// TIA Portal project "assembly_system" (V16)

(* hardware
DEVICE "ET 200SP station_1"  ET 200SP-Station
   slot 0: "IO device_1"  IM 155-6 PN/2 HF  6ES7 155-6AU01-0CN0  V4.2
   slot 0: "Rack_0"  Rack  6ES5 710-8MAx1
   slot 1: "DI 8x24VDC HF_1"  DI 8x24VDC HF  6ES7 131-6BF00-0CA0  V2.0
      slot 1: "DI 8x24VDC HF_1"  DI 8x24VDC HF
   slot 2: "DI 8x24VDC HF_2"  DI 8x24VDC HF  6ES7 131-6BF00-0CA0  V2.0
      slot 1: "DI 8x24VDC HF_2"  DI 8x24VDC HF
   slot 3: "DI 8x24VDC HF_3"  DI 8x24VDC HF  6ES7 131-6BF00-0CA0  V2.0
      slot 1: "DI 8x24VDC HF_3"  DI 8x24VDC HF
   slot 4: "DQ 8x24VDC/0.5A HF_1"  DQ 8x24VDC/0.5A HF  6ES7 132-6BF00-0CA0  V2.0
      slot 1: "DQ 8x24VDC/0.5A HF_1"  DQ 8x24VDC/0.5A HF
   slot 5: "DQ 8x24VDC/0.5A HF_2"  DQ 8x24VDC/0.5A HF  6ES7 132-6BF00-0CA0  V2.0
      slot 1: "DQ 8x24VDC/0.5A HF_2"  DQ 8x24VDC/0.5A HF
   slot 6: "Server module_1"  Server module  6ES7 193-6PA00-0AA0  V1.1
      slot 1: "Server module_1"  Server module
   slot 127: "BA 2xRJ45"  BA 2xRJ45  6ES7 193-6AR00-0AA0  V0.0
      slot 1: "Port_1"  X1 P1 R  6ES7 193-6AR00-0AA0  V0.0
      slot 2: "Port_2"  X1 P2 R  6ES7 193-6AR00-0AA0  V0.0
DEVICE "S7-1200 station_1"  S7-1200 Station
   slot 0: "Rack_0"  S7-1200 Rack  Rack  V1.0
   slot 1: "PLC_1"  CPU 1214C DC/DC/DC  6ES7 214-1AG40-0XB0  V4.4
DEVICE "SCALANCE X005"  SCALANCE X-Station
   slot 0: "Switch_1"  6GK5 005-0BA00-1AB2  V1.0
   slot 0: "SCALANCE X rack"  Rail
*)

// ===== PLC "PLC_1"  CPU 1214C DC/DC/DC =====

VAR_GLOBAL   // PLC tag table "Default tag table"
   "Tag_1" AT %M98.0 : Bool;
   "Tag_2" AT %M98.1 : Bool;
   "Tag_3" AT %M98.2 : Bool;
   "Clock_Byte" AT %MB200 : Byte;
   "Clock_10Hz" AT %M200.0 : Bool;
   "Clock_5Hz" AT %M200.1 : Bool;
   "Clock_2.5Hz" AT %M200.2 : Bool;
   "Clock_2Hz" AT %M200.3 : Bool;
   "Clock_1.25Hz" AT %M200.4 : Bool;
   "Clock_1Hz" AT %M200.5 : Bool;
   "Clock_0.625Hz" AT %M200.6 : Bool;
   "Clock_0.5Hz" AT %M200.7 : Bool;
   "Tag_4" AT %M10.6 : Bool;
   "System_Byte" AT %MB30 : Byte;
   "FirstScan" AT %M30.0 : Bool;
   "DiagStatusUpdate" AT %M30.1 : Bool;
   "AlwaysTRUE" AT %M30.2 : Bool;
   "AlwaysFALSE" AT %M30.3 : Bool;
END_VAR

VAR_GLOBAL   // PLC tag table "IO_TAGS"
   "START BUTTON  (N.O.) GAUGING" AT %I0.0 : Bool;
   "STOP BUTTON (N.C.) GAUGING" AT %I0.1 : Bool;
   "EMERGENCY STOP BUTTON (N.C.)" AT %I0.2 : Bool;
   "OUTPUT POWER ON (WHITE) GAUGING" AT %I0.3 : Bool;
   "INPUT 1 FROM PREVIOUS STATION GAUGING" AT %I0.4 : Bool;
   "RESET INDEXING STATION" AT %I0.5 : Bool;
   "AUTO INDEXNIG STATION" AT %I0.6 : Bool;
   "INPUT 2 FROM NEXT STATION GAUGING" AT %I0.7 : Bool;
   "RESET/AUTO SWITCH (RESET)" AT %I1.0 : Bool;
   "RESET/AUTO SWITCH (AUTO)" AT %I1.1 : Bool;
   "REJECT CYLINDER 3A RETRACTED GAUGING" AT %I1.2 : Bool;
   "REJECT CYLINDER 3A EXTENDED GAUGING" AT %I1.3 : Bool;
   "TRANSFER CYLINDER 1A RETRACTED GAUGING" AT %I1.4 : Bool;
   "TRANSFER CYLINDER 1A EXTENDED GAUGING" AT %I1.5 : Bool;
   "TRAVERSE IN END OF TRAVEL POSITION" AT %I4.6 : Bool;
   "TRAVERSE IN START OF TRAVEL POSITION" AT %I4.7 : Bool;
   "PART IN HEIGHT MEASURING POSITION" AT %I2.0 : Bool;
   "PART HEIGHT READING" AT %I2.1 : Bool;
   "GAUGING PORT NOT DETECTED (LIGHT SENSOR)" AT %I2.2 : Bool;
   "AUTOMATIC ON  LAMP (GREEN)" AT %Q0.0 : Bool;
   "OUTPUT 1 TO PREVIOUS STATION GAUGING" AT %Q0.1 : Bool;
   "OUTPUT 2 TO PREVIOUS STATION GAUGING" AT %Q0.2 : Bool;
   "OUTPUT 1 TO NEXT STATION GAUGING" AT %Q0.3 : Bool;
   "OUTPUT 2 TO NEXT STATION GAUGING" AT %Q0.4 : Bool;
   "EXTEND REJECT CYLINDER GAUGING" AT %Q0.5 : Bool;
   "EXTEND TRANSFER CYLINDER GAUGING" AT %Q0.6 : Bool;
   "RETRACT TRANSFER CYLINDER GAUGING" AT %Q0.7 : Bool;
   "GAUGING MOTOR STARTER FORWARD" AT %Q1.0 : Bool;
   "GAUGING MOTOR STARTER REVERSE" AT %Q1.1 : Bool;
   "EXTEND LIFT CYLINDER INDEXING" AT %Q3.6 : Bool;
   "AUTOMATIC ON (GREEN)(1)" AT %Q2.0 : Bool;
   "CLOSE GRIPPER 3A(1)" AT %Q3.3 : Bool;
   "EMERGENCY STOP BUTTON (N.C.) INDEXING" AT %I2.5 : Bool;
   "EXTEND LIFT CYLINDER 1A GAUGING" AT %Q2.6 : Bool;
   "EXTEND ROTATION CYLINDER 2A INDEXING" AT %Q3.4 : Bool;
   "EXTEND TRANSFER CYLINDER 3A INDEXING" AT %Q2.5 : Bool;
   "INDEXING TABLE IN HOME POSITION" AT %I4.3 : Bool;
   "INPUT 1 FROM NEXT STATION INDEXING" AT %I3.1 : Bool;
   "INPUT 1 FROM PREVIOUS STATION INDEXING" AT %I2.7 : Bool;
   "INPUT 2 FROM NEXT STATION INDEXING" AT %I3.2 : Bool;
   "INPUT 2 FROM PREVIOUS STATION INDEXING" AT %I3.0 : Bool;
   "LIFT CYLINDER 1A EXTENDED INDEXING" AT %I3.6 : Bool;
   "LIFT CYLINDER 1A RETRACTED INDEXING" AT %I3.5 : Bool;
   "OUTPUT 1 TO NEXT STATION INDEXING" AT %Q2.3 : Bool;
   "OUTPUT 1 TO PREVIOUS STATION INDEXING" AT %Q2.1 : Bool;
   "OUTPUT 2 TO NEXT STATION INDEXING" AT %Q2.4 : Bool;
   "OUTPUT 2 TO PREVIOUS STATION INDEXING" AT %Q2.2 : Bool;
   "OUTPUT POWER ON (WHITE) INDEXING" AT %I2.6 : Bool;
   "PART PRESENT (INITIAL POSITION)" AT %I4.5 : Bool;
   "PART PRESENT (ORIENTATION POSITION)" AT %I3.7 : Bool;
   "RELEASE GRIPPER 3A" AT %Q3.2 : Bool;
   "RETRACT LIFT CYLINDER 1A INDEXING" AT %Q2.7 : Bool;
   "RETRACT ROTATION CYLINDER 2A INDEXING" AT %Q3.5 : Bool;
   "ROTATION CYLINDER 2A EXTENDED INDEXING" AT %I4.1 : Bool;
   "ROTATION CYLINDER 2A RETRACTED INDEXING" AT %I4.0 : Bool;
   "INDEXING SPOOL UPPER PORT DETECTED" AT %I4.2 : Bool;
   "START BUTTON  (N.O.) INDEXING" AT %I2.3 : Bool;
   "STEPPER MOTOR  45°" AT %Q3.0 : Bool;
   "STEPPER MOTOR 90°" AT %Q3.1 : Bool;
   "STEPPER MOTOR READY" AT %I4.4 : Bool;
   "STOP BUTTON (N.C.) INDEXING" AT %I2.4 : Bool;
   "TRANSFER CYLINDER 4A EXTENDED(1)" AT %I3.4 : Bool;
   "TRANSFER CYLINDER 4A RETRACTED(1)" AT %I3.3 : Bool;
END_VAR

DATA_BLOCK "gauging_Modes_data"   // DB1
{ S7_Optimized_Access := 'TRUE' }
VERSION : 0.1
   VAR
      Automatic : Bool;
      Manual : Bool;
      Reset : Bool;
      "Pre-Automatic" : Bool;
   END_VAR
BEGIN
END_DATA_BLOCK

DATA_BLOCK "gauging_outputs_data"   // DB2
{ S7_Optimized_Access := 'TRUE' }
VERSION : 0.1
   VAR
      "Extend reject cylinder" : Bool;
      "Extend transfer cylinder" : Bool;
      "Retract transfer cylinder" : Bool;
      "Motor forward" : Bool;
      "Motor Reverse" : Bool;
      "Extend Lift Cylinder" : Bool;
      Output : Bool;
   END_VAR
BEGIN
END_DATA_BLOCK

DATA_BLOCK "gauging_status_data"   // DB3
{ S7_Optimized_Access := 'TRUE' }
VERSION : 0.1
   VAR
      steps : Int;
      "port not detected" : Bool;
      "height detected" : Bool;
      next_step : Bool;
      input_from_previous_Station : Bool;
   END_VAR
BEGIN
END_DATA_BLOCK

DATA_BLOCK "indexing_Modes_data"   // DB18
{ S7_Optimized_Access := 'TRUE' }
VERSION : 0.1
   VAR
      Automatic : Bool;
      Manual : Bool;
      Reset : Bool;
      "Pre-Automatic" : Bool;
   END_VAR
BEGIN
END_DATA_BLOCK

DATA_BLOCK "indexing_output_data"   // DB19
{ S7_Optimized_Access := 'TRUE' }
VERSION : 0.1
   VAR
      "extend transfer cylinder" : Bool;
      "extend lift cylinder_1" : Bool;
      "extend lift cylinder_2" : Bool;
      "retract lift cylinder_1" : Bool;
      "retract lift cylinder_2" : Bool;
      STEP1_MOTOR_45 : Bool;
      STEP3_MOTOR_45 : Bool;
      STEP4_MOTOR_90 : Bool;
      STEP11_MOTOR_90 : Bool;
      "release gripper" : Bool;
      "close gripper" : Bool;
      "extend rotation" : Bool;
      "retract rotation" : Bool;
      output : Bool;
   END_VAR
BEGIN
END_DATA_BLOCK

DATA_BLOCK "indexing_status_data"   // DB20
{ S7_Optimized_Access := 'TRUE' }
VERSION : 0.1
   VAR
      "CORRECT ORIENTATION" : Bool;
      STEPS : Int;
      next_step : Bool;
      previous_output : Bool;
   END_VAR
BEGIN
END_DATA_BLOCK

// folder: System blocks/Program resources

DATA_BLOCK "port_detection_wait"   // DB4
{ S7_Optimized_Access := 'TRUE' }
AUTHOR : Simatic
FAMILY : IEC
NAME : IEC_TMR
VERSION : 1.0
// stored: InstanceOfName IEC_TIMER
"IEC_TIMER"
BEGIN
END_DATA_BLOCK

DATA_BLOCK "retract_delay"   // DB5
{ S7_Optimized_Access := 'TRUE' }
AUTHOR : Simatic
FAMILY : IEC
NAME : IEC_TMR
VERSION : 1.0
// stored: InstanceOfName IEC_TIMER
"IEC_TIMER"
BEGIN
END_DATA_BLOCK

DATA_BLOCK "next_step_delay"   // DB6
{ S7_Optimized_Access := 'TRUE' }
AUTHOR : Simatic
FAMILY : IEC
NAME : IEC_TMR
VERSION : 1.0
// stored: InstanceOfName IEC_TIMER
"IEC_TIMER"
BEGIN
END_DATA_BLOCK

DATA_BLOCK "height_Timer_0_DB"   // DB7
{ S7_Optimized_Access := 'TRUE' }
AUTHOR : Simatic
FAMILY : IEC
NAME : IEC_TMR
VERSION : 1.0
// stored: InstanceOfName IEC_TIMER
"IEC_TIMER"
BEGIN
END_DATA_BLOCK

DATA_BLOCK "retract_wait"   // DB8
{ S7_Optimized_Access := 'TRUE' }
AUTHOR : Simatic
FAMILY : IEC
NAME : IEC_TMR
VERSION : 1.0
// stored: InstanceOfName IEC_TIMER
"IEC_TIMER"
BEGIN
END_DATA_BLOCK

DATA_BLOCK "next_step_wait_1"   // DB9
{ S7_Optimized_Access := 'TRUE' }
AUTHOR : Simatic
FAMILY : IEC
NAME : IEC_TMR
VERSION : 1.0
// stored: InstanceOfName IEC_TIMER
"IEC_TIMER"
BEGIN
END_DATA_BLOCK

DATA_BLOCK "motor_wait"   // DB10
{ S7_Optimized_Access := 'TRUE' }
AUTHOR : Simatic
FAMILY : IEC
NAME : IEC_TMR
VERSION : 1.0
// stored: InstanceOfName IEC_TIMER
"IEC_TIMER"
BEGIN
END_DATA_BLOCK

DATA_BLOCK "extend_retract_wait"   // DB11
{ S7_Optimized_Access := 'TRUE' }
AUTHOR : Simatic
FAMILY : IEC
NAME : IEC_TMR
VERSION : 1.0
// stored: InstanceOfName IEC_TIMER
"IEC_TIMER"
BEGIN
END_DATA_BLOCK

DATA_BLOCK "wait_Timer"   // DB12
{ S7_Optimized_Access := 'TRUE' }
AUTHOR : Simatic
FAMILY : IEC
NAME : IEC_TMR
VERSION : 1.0
// stored: InstanceOfName IEC_TIMER
"IEC_TIMER"
BEGIN
END_DATA_BLOCK

DATA_BLOCK "motor90_Timer"   // DB13
{ S7_Optimized_Access := 'TRUE' }
AUTHOR : Simatic
FAMILY : IEC
NAME : IEC_TMR
VERSION : 1.0
// stored: InstanceOfName IEC_TIMER
"IEC_TIMER"
BEGIN
END_DATA_BLOCK

DATA_BLOCK "delay_gripper_clamp"   // DB14
{ S7_Optimized_Access := 'TRUE' }
AUTHOR : Simatic
FAMILY : IEC
NAME : IEC_TMR
VERSION : 1.0
// stored: InstanceOfName IEC_TIMER
"IEC_TIMER"
BEGIN
END_DATA_BLOCK

DATA_BLOCK "lift_wait_DB"   // DB15
{ S7_Optimized_Access := 'TRUE' }
AUTHOR : Simatic
FAMILY : IEC
NAME : IEC_TMR
VERSION : 1.0
// stored: InstanceOfName IEC_TIMER
"IEC_TIMER"
BEGIN
END_DATA_BLOCK

DATA_BLOCK "gripper_Timer"   // DB16
{ S7_Optimized_Access := 'TRUE' }
AUTHOR : Simatic
FAMILY : IEC
NAME : IEC_TMR
VERSION : 1.0
// stored: InstanceOfName IEC_TIMER
"IEC_TIMER"
BEGIN
END_DATA_BLOCK

DATA_BLOCK "transfer_delay_DB"   // DB17
{ S7_Optimized_Access := 'TRUE' }
AUTHOR : Simatic
FAMILY : IEC
NAME : IEC_TMR
VERSION : 1.0
// stored: InstanceOfName IEC_TIMER
"IEC_TIMER"
BEGIN
END_DATA_BLOCK

DATA_BLOCK "retract_delay_1"   // DB21
{ S7_Optimized_Access := 'TRUE' }
AUTHOR : Simatic
FAMILY : IEC
NAME : IEC_TMR
VERSION : 1.0
// stored: InstanceOfName IEC_TIMER
"IEC_TIMER"
BEGIN
END_DATA_BLOCK

DATA_BLOCK "retract_DB"   // DB22
{ S7_Optimized_Access := 'TRUE' }
AUTHOR : Simatic
FAMILY : IEC
NAME : IEC_TMR
VERSION : 1.0
// stored: InstanceOfName IEC_TIMER
"IEC_TIMER"
BEGIN
END_DATA_BLOCK

// folder: (top level)

FUNCTION "gauging_modes" : Void   // FC1, LAD
TITLE = Modes Setup
{ S7_Optimized_Access := 'TRUE' }
VERSION : 0.1
BEGIN

REGION Network 1: Automatic Mode
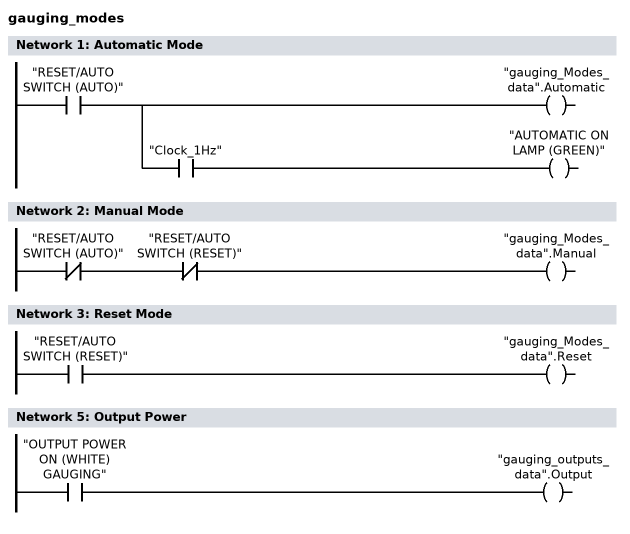
   RUNG wire#powerrail
      Contact( "RESET/AUTO SWITCH (AUTO)" )
      wire#w1
      Coil( "gauging_Modes_data".Automatic )
   END_RUNG
   RUNG wire#w1
      Contact( "Clock_1Hz" )
      Coil( "AUTOMATIC ON  LAMP (GREEN)" )
   END_RUNG
   // the same network as SCL:
   "gauging_Modes_data".Automatic := "RESET/AUTO SWITCH (AUTO)";
   "AUTOMATIC ON  LAMP (GREEN)" := "RESET/AUTO SWITCH (AUTO)" AND "Clock_1Hz";
END_REGION

REGION Network 2: Manual Mode
   RUNG wire#powerrail
      I_Contact( "RESET/AUTO SWITCH (AUTO)" )
      I_Contact( "RESET/AUTO SWITCH (RESET)" )
      Coil( "gauging_Modes_data".Manual )
   END_RUNG
   // the same network as SCL:
   "gauging_Modes_data".Manual := NOT "RESET/AUTO SWITCH (AUTO)" AND NOT "RESET/AUTO SWITCH (RESET)";
END_REGION

REGION Network 3: Reset Mode
   RUNG wire#powerrail
      Contact( "RESET/AUTO SWITCH (RESET)" )
      Coil( "gauging_Modes_data".Reset )
   END_RUNG
   // the same network as SCL:
   "gauging_Modes_data".Reset := "RESET/AUTO SWITCH (RESET)";
END_REGION

REGION Network 4: Pre-Automatic Mode
END_REGION

REGION Network 5: Output Power
   RUNG wire#powerrail
      Contact( "OUTPUT POWER ON (WHITE) GAUGING" )
      Coil( "gauging_outputs_data".Output )
   END_RUNG
   // the same network as SCL:
   "gauging_outputs_data".Output := "OUTPUT POWER ON (WHITE) GAUGING";
END_REGION
END_FUNCTION

FUNCTION "gauging_outputs" : Void   // FC2, LAD
{ S7_Optimized_Access := 'TRUE' }
VERSION : 0.1
BEGIN

REGION Network 1: Gauging Reject Cylinder
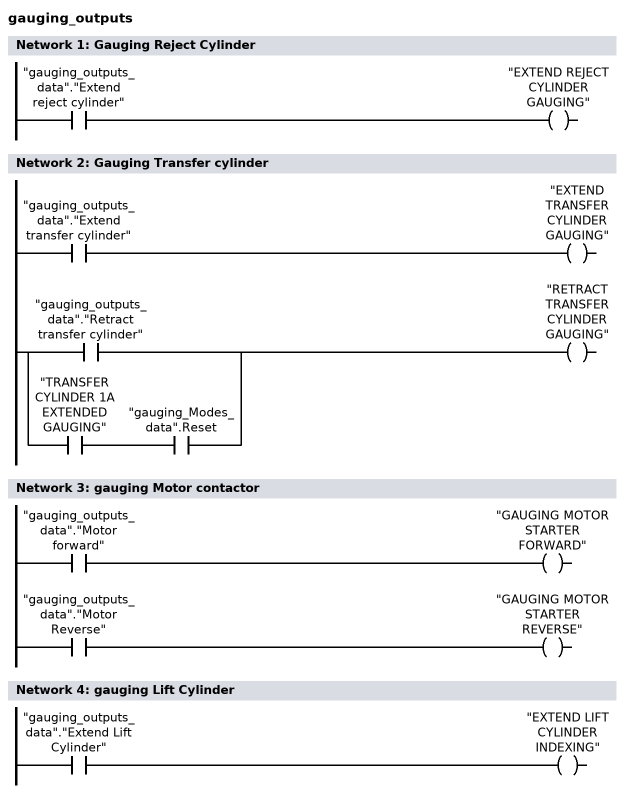
   RUNG wire#powerrail
      Contact( "gauging_outputs_data"."Extend reject cylinder" )
      Coil( "EXTEND REJECT CYLINDER GAUGING" )
   END_RUNG
   // the same network as SCL:
   "EXTEND REJECT CYLINDER GAUGING" := "gauging_outputs_data"."Extend reject cylinder";
END_REGION

REGION Network 2: Gauging Transfer cylinder
   RUNG wire#powerrail
      Contact( "gauging_outputs_data"."Extend transfer cylinder" )
      Coil( "EXTEND TRANSFER CYLINDER GAUGING" )
   END_RUNG
   RUNG wire#powerrail
      Contact( "gauging_outputs_data"."Retract transfer cylinder" )
      wire#w1
      Coil( "RETRACT TRANSFER CYLINDER GAUGING" )
   END_RUNG
   RUNG wire#powerrail
      Contact( "TRANSFER CYLINDER 1A EXTENDED GAUGING" )
      Contact( "gauging_Modes_data".Reset )
   END_RUNG wire#w1
   // the same network as SCL:
   "EXTEND TRANSFER CYLINDER GAUGING" := "gauging_outputs_data"."Extend transfer cylinder";
   "RETRACT TRANSFER CYLINDER GAUGING" := "gauging_outputs_data"."Retract transfer cylinder" OR ("TRANSFER CYLINDER 1A EXTENDED GAUGING" AND "gauging_Modes_data".Reset);
END_REGION

REGION Network 3: gauging Motor contactor
   RUNG wire#powerrail
      Contact( "gauging_outputs_data"."Motor forward" )
      Coil( "GAUGING MOTOR STARTER FORWARD" )
   END_RUNG
   RUNG wire#powerrail
      Contact( "gauging_outputs_data"."Motor Reverse" )
      Coil( "GAUGING MOTOR STARTER REVERSE" )
   END_RUNG
   // the same network as SCL:
   "GAUGING MOTOR STARTER FORWARD" := "gauging_outputs_data"."Motor forward";
   "GAUGING MOTOR STARTER REVERSE" := "gauging_outputs_data"."Motor Reverse";
END_REGION

REGION Network 4: gauging Lift Cylinder
   RUNG wire#powerrail
      Contact( "gauging_outputs_data"."Extend Lift Cylinder" )
      Coil( "EXTEND LIFT CYLINDER INDEXING" )
   END_RUNG
   // the same network as SCL:
   "EXTEND LIFT CYLINDER INDEXING" := "gauging_outputs_data"."Extend Lift Cylinder";
END_REGION
END_FUNCTION

FUNCTION "gauging_utils" : Void   // FC3, LAD
{ S7_Optimized_Access := 'TRUE' }
VERSION : 0.1
   VAR_TEMP   // added for the SCL form of the ladder/FBD networks
      _w1 : Bool;
      _w2 : Bool;
   END_VAR
BEGIN

REGION Network 1: SETUP: output, start, reset
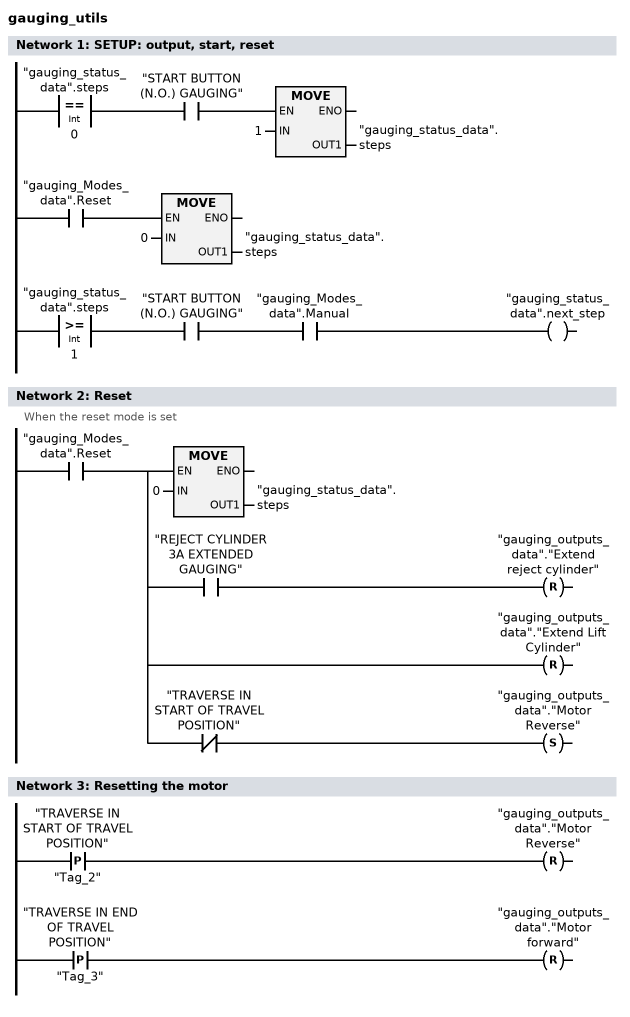
   RUNG wire#powerrail
      { S7_Templates := "SrcType := Int" } EQ_Contact(in1 := "gauging_status_data".steps, in2 := 0)
      Contact( "START BUTTON  (N.O.) GAUGING" )
      Move(in := 1, out1 => "gauging_status_data".steps)
   END_RUNG
   RUNG wire#powerrail
      Contact( "gauging_Modes_data".Reset )
      Move(in := 0, out1 => "gauging_status_data".steps)
   END_RUNG
   RUNG wire#powerrail
      { S7_Templates := "SrcType := Int" } GE_Contact(in1 := "gauging_status_data".steps, in2 := 1)
      Contact( "START BUTTON  (N.O.) GAUGING" )
      Contact( "gauging_Modes_data".Manual )
      Coil( "gauging_status_data".next_step )
   END_RUNG
   // the same network as SCL:
   IF ("gauging_status_data".steps = 0) AND "START BUTTON  (N.O.) GAUGING" THEN
       "gauging_status_data".steps := 1;
   END_IF;
   IF "gauging_Modes_data".Reset THEN "gauging_status_data".steps := 0; END_IF;
   "gauging_status_data".next_step := ("gauging_status_data".steps >= 1) AND "START BUTTON  (N.O.) GAUGING" AND "gauging_Modes_data".Manual;
END_REGION

REGION Network 2: Reset
   // When the reset mode is set
   RUNG wire#powerrail
      Contact( "gauging_Modes_data".Reset )
      wire#w1
      Move(in := 0, out1 => "gauging_status_data".steps)
   END_RUNG
   RUNG wire#w1
      Contact( "REJECT CYLINDER 3A EXTENDED GAUGING" )
      R_Coil( "gauging_outputs_data"."Extend reject cylinder" )
   END_RUNG
   RUNG wire#w1
      R_Coil( "gauging_outputs_data"."Extend Lift Cylinder" )
   END_RUNG
   RUNG wire#w1
      I_Contact( "TRAVERSE IN START OF TRAVEL POSITION" )
      S_Coil( "gauging_outputs_data"."Motor Reverse" )
   END_RUNG
   // the same network as SCL:
   IF "gauging_Modes_data".Reset THEN "gauging_status_data".steps := 0; END_IF;
   IF "gauging_Modes_data".Reset AND "REJECT CYLINDER 3A EXTENDED GAUGING" THEN
       "gauging_outputs_data"."Extend reject cylinder" := FALSE;
   END_IF;
   IF "gauging_Modes_data".Reset THEN "gauging_outputs_data"."Extend Lift Cylinder" := FALSE; END_IF;
   IF "gauging_Modes_data".Reset AND NOT "TRAVERSE IN START OF TRAVEL POSITION" THEN
       "gauging_outputs_data"."Motor Reverse" := TRUE;
   END_IF;
END_REGION

REGION Network 3: Resetting the motor
   RUNG wire#powerrail
      P_Contact(operand := "TRAVERSE IN START OF TRAVEL POSITION", bit := "Tag_2")
      R_Coil( "gauging_outputs_data"."Motor Reverse" )
   END_RUNG
   RUNG wire#powerrail
      P_Contact(operand := "TRAVERSE IN END OF TRAVEL POSITION", bit := "Tag_3")
      R_Coil( "gauging_outputs_data"."Motor forward" )
   END_RUNG
   // the same network as SCL:
   #_w1 := "TRAVERSE IN START OF TRAVEL POSITION" AND NOT "Tag_2";   // rising edge of "TRAVERSE IN START OF TRAVEL POSITION"
   "Tag_2" := "TRAVERSE IN START OF TRAVEL POSITION";
   IF #_w1 THEN "gauging_outputs_data"."Motor Reverse" := FALSE; END_IF;
   #_w2 := "TRAVERSE IN END OF TRAVEL POSITION" AND NOT "Tag_3";   // rising edge of "TRAVERSE IN END OF TRAVEL POSITION"
   "Tag_3" := "TRAVERSE IN END OF TRAVEL POSITION";
   IF #_w2 THEN "gauging_outputs_data"."Motor forward" := FALSE; END_IF;
END_REGION
END_FUNCTION

FUNCTION "gauging_operation" : Void   // FC4, LAD
{ S7_Optimized_Access := 'TRUE' }
VERSION : 0.1
   VAR_TEMP   // added for the SCL form of the ladder/FBD networks
      _w1 : Bool;
   END_VAR
BEGIN

REGION Network 1: Setup
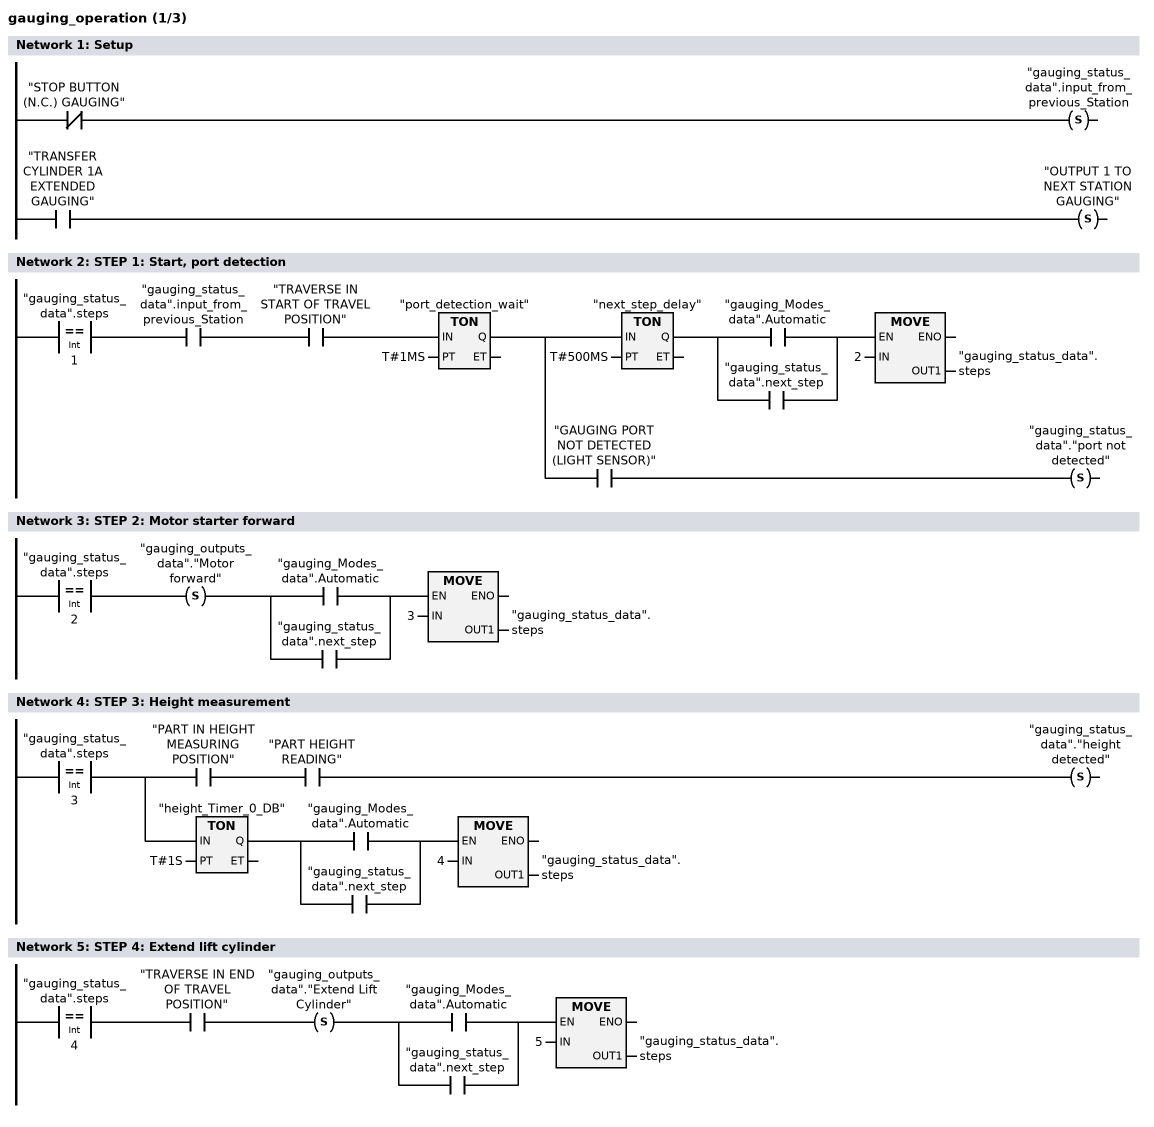
   RUNG wire#powerrail
      I_Contact( "STOP BUTTON (N.C.) GAUGING" )
      S_Coil( "gauging_status_data".input_from_previous_Station )
   END_RUNG
   RUNG wire#powerrail
      Contact( "TRANSFER CYLINDER 1A EXTENDED GAUGING" )
      S_Coil( "OUTPUT 1 TO NEXT STATION GAUGING" )
   END_RUNG
   // the same network as SCL:
   IF NOT "STOP BUTTON (N.C.) GAUGING" THEN
       "gauging_status_data".input_from_previous_Station := TRUE;
   END_IF;
   IF "TRANSFER CYLINDER 1A EXTENDED GAUGING" THEN "OUTPUT 1 TO NEXT STATION GAUGING" := TRUE; END_IF;
END_REGION

REGION Network 2: STEP 1: Start, port detection
   "port_detection_wait".TON(IN := ("gauging_status_data".steps = 1) AND "gauging_status_data".input_from_previous_Station AND "TRAVERSE IN START OF TRAVEL POSITION",
                           PT := T#1MS);
   "next_step_delay".TON(IN := "port_detection_wait".Q, PT := T#500MS);
   IF "next_step_delay".Q AND ("gauging_Modes_data".Automatic OR "gauging_status_data".next_step) THEN
       "gauging_status_data".steps := 2;
   END_IF;
   IF "port_detection_wait".Q AND "GAUGING PORT NOT DETECTED (LIGHT SENSOR)" THEN
       "gauging_status_data"."port not detected" := TRUE;
   END_IF;
END_REGION

REGION Network 3: STEP 2: Motor starter forward
   RUNG wire#powerrail
      { S7_Templates := "SrcType := Int" } EQ_Contact(in1 := "gauging_status_data".steps, in2 := 2)
      S_Coil( "gauging_outputs_data"."Motor forward" )
      wire#w1
      Contact( "gauging_Modes_data".Automatic )
      wire#w2
      Move(in := 3, out1 => "gauging_status_data".steps)
   END_RUNG
   RUNG wire#w1
      Contact( "gauging_status_data".next_step )
   END_RUNG wire#w2
   // the same network as SCL:
   #_w1 := "gauging_status_data".steps = 2;
   IF #_w1 THEN "gauging_outputs_data"."Motor forward" := TRUE; END_IF;
   IF #_w1 AND ("gauging_Modes_data".Automatic OR "gauging_status_data".next_step) THEN
       "gauging_status_data".steps := 3;
   END_IF;
END_REGION

REGION Network 4: STEP 3: Height measurement
   #_w1 := "gauging_status_data".steps = 3;
   IF #_w1 AND "PART IN HEIGHT MEASURING POSITION" AND "PART HEIGHT READING" THEN
       "gauging_status_data"."height detected" := TRUE;
   END_IF;
   "height_Timer_0_DB".TON(IN := #_w1, PT := T#1S);
   IF "height_Timer_0_DB".Q AND ("gauging_Modes_data".Automatic OR "gauging_status_data".next_step) THEN
       "gauging_status_data".steps := 4;
   END_IF;
END_REGION

REGION Network 5: STEP 4: Extend lift cylinder
   RUNG wire#powerrail
      { S7_Templates := "SrcType := Int" } EQ_Contact(in1 := "gauging_status_data".steps, in2 := 4)
      Contact( "TRAVERSE IN END OF TRAVEL POSITION" )
      S_Coil( "gauging_outputs_data"."Extend Lift Cylinder" )
      wire#w1
      Contact( "gauging_Modes_data".Automatic )
      wire#w2
      Move(in := 5, out1 => "gauging_status_data".steps)
   END_RUNG
   RUNG wire#w1
      Contact( "gauging_status_data".next_step )
   END_RUNG wire#w2
   // the same network as SCL:
   #_w1 := ("gauging_status_data".steps = 4) AND "TRAVERSE IN END OF TRAVEL POSITION";
   IF #_w1 THEN "gauging_outputs_data"."Extend Lift Cylinder" := TRUE; END_IF;
   IF #_w1 AND ("gauging_Modes_data".Automatic OR "gauging_status_data".next_step) THEN
       "gauging_status_data".steps := 5;
   END_IF;
END_REGION

REGION Network 6: STEP 5: Check port and height orientation
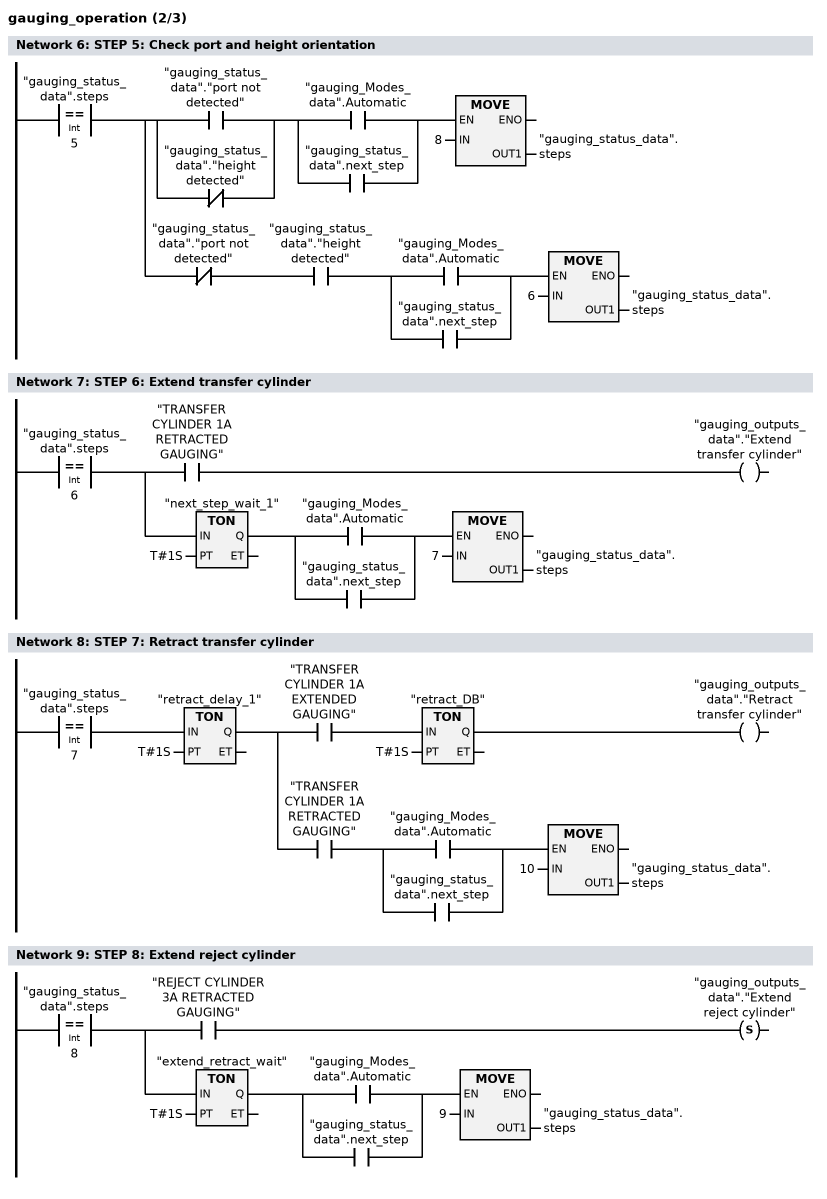
   RUNG wire#powerrail
      { S7_Templates := "SrcType := Int" } EQ_Contact(in1 := "gauging_status_data".steps, in2 := 5)
      wire#w1
      Contact( "gauging_status_data"."port not detected" )
      wire#w2
      Contact( "gauging_Modes_data".Automatic )
      wire#w3
      Move(in := 8, out1 => "gauging_status_data".steps)
   END_RUNG
   RUNG wire#w1
      I_Contact( "gauging_status_data"."height detected" )
   END_RUNG wire#w2
   RUNG wire#w2
      Contact( "gauging_status_data".next_step )
   END_RUNG wire#w3
   RUNG wire#w1
      I_Contact( "gauging_status_data"."port not detected" )
      Contact( "gauging_status_data"."height detected" )
      wire#w4
      Contact( "gauging_Modes_data".Automatic )
      wire#w5
      Move(in := 6, out1 => "gauging_status_data".steps)
   END_RUNG
   RUNG wire#w4
      Contact( "gauging_status_data".next_step )
   END_RUNG wire#w5
   // the same network as SCL:
   #_w1 := "gauging_status_data".steps = 5;
   IF #_w1 AND ("gauging_status_data"."port not detected" OR NOT "gauging_status_data"."height detected") AND ("gauging_Modes_data".Automatic OR "gauging_status_data".next_step) THEN
       "gauging_status_data".steps := 8;
   END_IF;
   IF #_w1 AND NOT "gauging_status_data"."port not detected" AND "gauging_status_data"."height detected" AND ("gauging_Modes_data".Automatic OR "gauging_status_data".next_step) THEN
       "gauging_status_data".steps := 6;
   END_IF;
END_REGION

REGION Network 7: STEP 6: Extend transfer cylinder
   #_w1 := "gauging_status_data".steps = 6;
   "gauging_outputs_data"."Extend transfer cylinder" := #_w1 AND "TRANSFER CYLINDER 1A RETRACTED GAUGING";
   "next_step_wait_1".TON(IN := #_w1, PT := T#1S);
   IF "next_step_wait_1".Q AND ("gauging_Modes_data".Automatic OR "gauging_status_data".next_step) THEN
       "gauging_status_data".steps := 7;
   END_IF;
END_REGION

REGION Network 8: STEP 7: Retract transfer cylinder
   "retract_delay_1".TON(IN := "gauging_status_data".steps = 7, PT := T#1S);
   "retract_DB".TON(IN := "retract_delay_1".Q AND "TRANSFER CYLINDER 1A EXTENDED GAUGING", PT := T#1S);
   "gauging_outputs_data"."Retract transfer cylinder" := "retract_DB".Q;
   IF "retract_delay_1".Q AND "TRANSFER CYLINDER 1A RETRACTED GAUGING" AND ("gauging_Modes_data".Automatic OR "gauging_status_data".next_step) THEN
       "gauging_status_data".steps := 10;
   END_IF;
END_REGION

REGION Network 9: STEP 8: Extend reject cylinder
   #_w1 := "gauging_status_data".steps = 8;
   IF #_w1 AND "REJECT CYLINDER 3A RETRACTED GAUGING" THEN
       "gauging_outputs_data"."Extend reject cylinder" := TRUE;
   END_IF;
   "extend_retract_wait".TON(IN := #_w1, PT := T#1S);
   IF "extend_retract_wait".Q AND ("gauging_Modes_data".Automatic OR "gauging_status_data".next_step) THEN
       "gauging_status_data".steps := 9;
   END_IF;
END_REGION

REGION Network 10: STEP 9: Retract reject cylinder
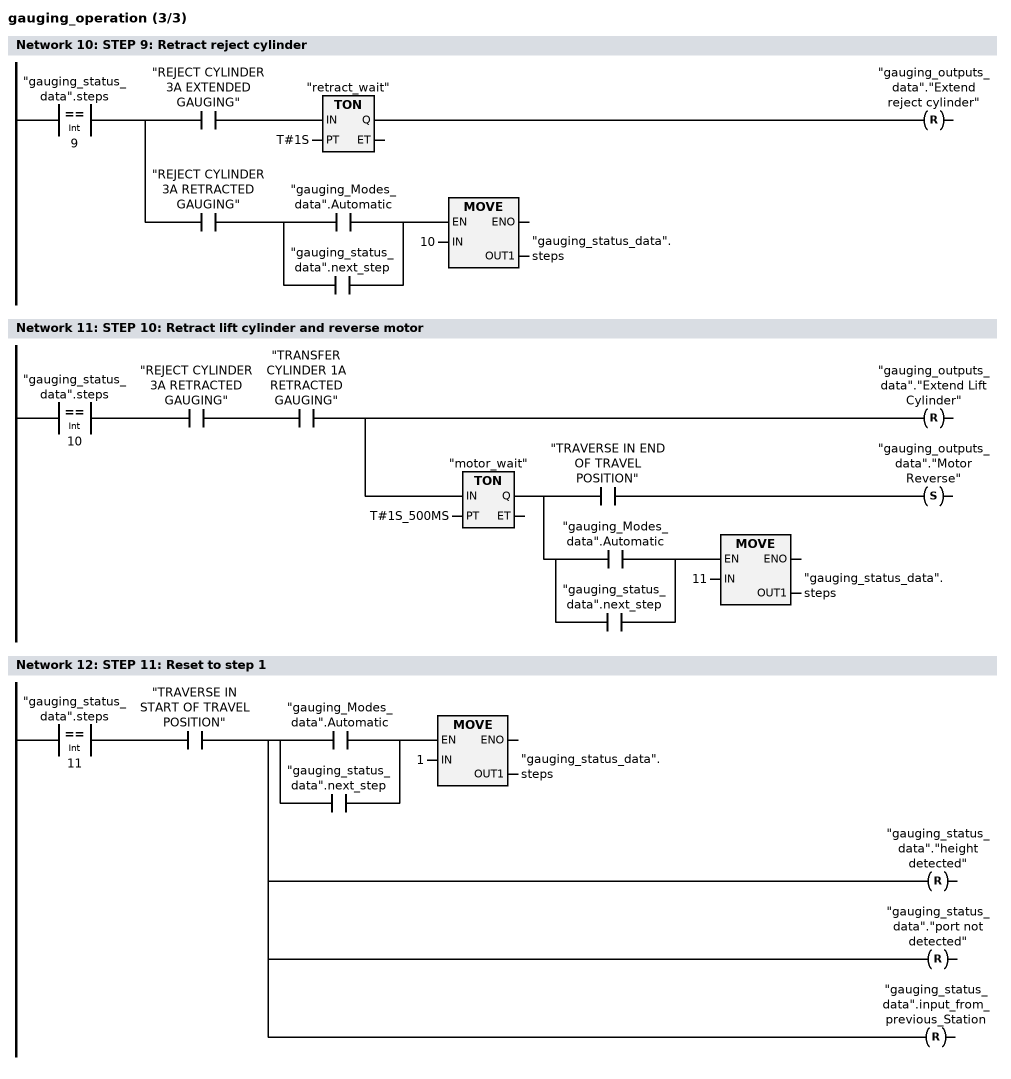
   #_w1 := "gauging_status_data".steps = 9;
   "retract_wait".TON(IN := #_w1 AND "REJECT CYLINDER 3A EXTENDED GAUGING", PT := T#1S);
   IF "retract_wait".Q THEN "gauging_outputs_data"."Extend reject cylinder" := FALSE; END_IF;
   IF #_w1 AND "REJECT CYLINDER 3A RETRACTED GAUGING" AND ("gauging_Modes_data".Automatic OR "gauging_status_data".next_step) THEN
       "gauging_status_data".steps := 10;
   END_IF;
END_REGION

REGION Network 11: STEP 10: Retract lift cylinder and reverse motor
   #_w1 := ("gauging_status_data".steps = 10) AND "REJECT CYLINDER 3A RETRACTED GAUGING" AND "TRANSFER CYLINDER 1A RETRACTED GAUGING";
   IF #_w1 THEN "gauging_outputs_data"."Extend Lift Cylinder" := FALSE; END_IF;
   "motor_wait".TON(IN := #_w1, PT := T#1S_500MS);
   IF "motor_wait".Q AND "TRAVERSE IN END OF TRAVEL POSITION" THEN
       "gauging_outputs_data"."Motor Reverse" := TRUE;
   END_IF;
   IF "motor_wait".Q AND ("gauging_Modes_data".Automatic OR "gauging_status_data".next_step) THEN
       "gauging_status_data".steps := 11;
   END_IF;
END_REGION

REGION Network 12: STEP 11: Reset to step 1
   RUNG wire#powerrail
      { S7_Templates := "SrcType := Int" } EQ_Contact(in1 := "gauging_status_data".steps, in2 := 11)
      Contact( "TRAVERSE IN START OF TRAVEL POSITION" )
      wire#w1
      Contact( "gauging_Modes_data".Automatic )
      wire#w2
      Move(in := 1, out1 => "gauging_status_data".steps)
   END_RUNG
   RUNG wire#w1
      Contact( "gauging_status_data".next_step )
   END_RUNG wire#w2
   RUNG wire#w1
      R_Coil( "gauging_status_data"."height detected" )
   END_RUNG
   RUNG wire#w1
      R_Coil( "gauging_status_data"."port not detected" )
   END_RUNG
   RUNG wire#w1
      R_Coil( "gauging_status_data".input_from_previous_Station )
   END_RUNG
   // the same network as SCL:
   #_w1 := ("gauging_status_data".steps = 11) AND "TRAVERSE IN START OF TRAVEL POSITION";
   IF #_w1 AND ("gauging_Modes_data".Automatic OR "gauging_status_data".next_step) THEN
       "gauging_status_data".steps := 1;
   END_IF;
   IF #_w1 THEN
       "gauging_status_data"."height detected" := FALSE;
       "gauging_status_data"."port not detected" := FALSE;
       "gauging_status_data".input_from_previous_Station := FALSE;
   END_IF;
END_REGION
END_FUNCTION

FUNCTION "indexing_modes" : Void   // FC5, LAD
TITLE = Modes Setup
{ S7_Optimized_Access := 'TRUE' }
VERSION : 0.1
BEGIN

REGION Network 1: Automatic Mode
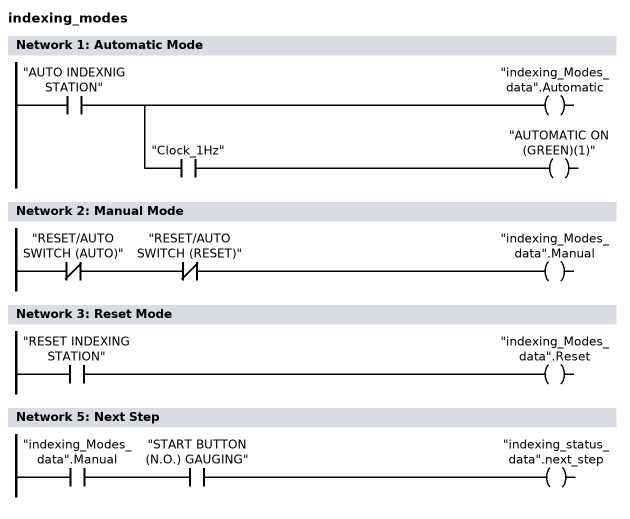
   RUNG wire#powerrail
      Contact( "AUTO INDEXNIG STATION" )
      wire#w1
      Coil( "indexing_Modes_data".Automatic )
   END_RUNG
   RUNG wire#w1
      Contact( "Clock_1Hz" )
      Coil( "AUTOMATIC ON (GREEN)(1)" )
   END_RUNG
   // the same network as SCL:
   "indexing_Modes_data".Automatic := "AUTO INDEXNIG STATION";
   "AUTOMATIC ON (GREEN)(1)" := "AUTO INDEXNIG STATION" AND "Clock_1Hz";
END_REGION

REGION Network 2: Manual Mode
   RUNG wire#powerrail
      I_Contact( "RESET/AUTO SWITCH (AUTO)" )
      I_Contact( "RESET/AUTO SWITCH (RESET)" )
      Coil( "indexing_Modes_data".Manual )
   END_RUNG
   // the same network as SCL:
   "indexing_Modes_data".Manual := NOT "RESET/AUTO SWITCH (AUTO)" AND NOT "RESET/AUTO SWITCH (RESET)";
END_REGION

REGION Network 3: Reset Mode
   RUNG wire#powerrail
      Contact( "RESET INDEXING STATION" )
      Coil( "indexing_Modes_data".Reset )
   END_RUNG
   // the same network as SCL:
   "indexing_Modes_data".Reset := "RESET INDEXING STATION";
END_REGION

REGION Network 4: Pre-Automatic Mode
END_REGION

REGION Network 5: Next Step
   RUNG wire#powerrail
      Contact( "indexing_Modes_data".Manual )
      Contact( "START BUTTON  (N.O.) GAUGING" )
      Coil( "indexing_status_data".next_step )
   END_RUNG
   // the same network as SCL:
   "indexing_status_data".next_step := "indexing_Modes_data".Manual AND "START BUTTON  (N.O.) GAUGING";
END_REGION
END_FUNCTION

FUNCTION "indexing_outputs" : Void   // FC6, LAD
{ S7_Optimized_Access := 'TRUE' }
VERSION : 0.1
BEGIN

REGION Network 1: indexing Transfer Cylinder
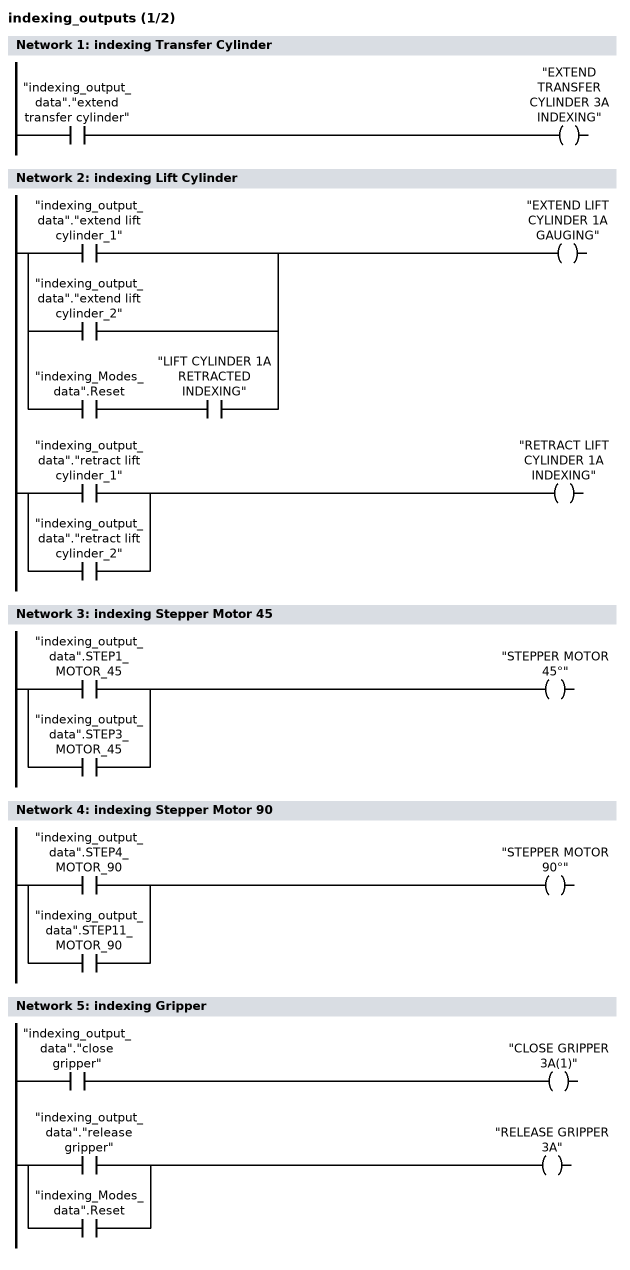
   RUNG wire#powerrail
      Contact( "indexing_output_data"."extend transfer cylinder" )
      Coil( "EXTEND TRANSFER CYLINDER 3A INDEXING" )
   END_RUNG
   // the same network as SCL:
   "EXTEND TRANSFER CYLINDER 3A INDEXING" := "indexing_output_data"."extend transfer cylinder";
END_REGION

REGION Network 2: indexing Lift Cylinder
   RUNG wire#powerrail
      Contact( "indexing_output_data"."extend lift cylinder_1" )
      wire#w1
      Coil( "EXTEND LIFT CYLINDER 1A GAUGING" )
   END_RUNG
   RUNG wire#powerrail
      Contact( "indexing_output_data"."extend lift cylinder_2" )
   END_RUNG wire#w1
   RUNG wire#powerrail
      Contact( "indexing_Modes_data".Reset )
      Contact( "LIFT CYLINDER 1A RETRACTED INDEXING" )
   END_RUNG wire#w1
   RUNG wire#powerrail
      Contact( "indexing_output_data"."retract lift cylinder_1" )
      wire#w2
      Coil( "RETRACT LIFT CYLINDER 1A INDEXING" )
   END_RUNG
   RUNG wire#powerrail
      Contact( "indexing_output_data"."retract lift cylinder_2" )
   END_RUNG wire#w2
   // the same network as SCL:
   "EXTEND LIFT CYLINDER 1A GAUGING" := "indexing_output_data"."extend lift cylinder_1" OR "indexing_output_data"."extend lift cylinder_2" OR ("indexing_Modes_data".Reset AND "LIFT CYLINDER 1A RETRACTED INDEXING");
   "RETRACT LIFT CYLINDER 1A INDEXING" := "indexing_output_data"."retract lift cylinder_1" OR "indexing_output_data"."retract lift cylinder_2";
END_REGION

REGION Network 3: indexing Stepper Motor 45
   RUNG wire#powerrail
      Contact( "indexing_output_data".STEP1_MOTOR_45 )
      wire#w1
      Coil( "STEPPER MOTOR  45°" )
   END_RUNG
   RUNG wire#powerrail
      Contact( "indexing_output_data".STEP3_MOTOR_45 )
   END_RUNG wire#w1
   // the same network as SCL:
   "STEPPER MOTOR  45°" := "indexing_output_data".STEP1_MOTOR_45 OR "indexing_output_data".STEP3_MOTOR_45;
END_REGION

REGION Network 4: indexing Stepper Motor 90
   RUNG wire#powerrail
      Contact( "indexing_output_data".STEP4_MOTOR_90 )
      wire#w1
      Coil( "STEPPER MOTOR 90°" )
   END_RUNG
   RUNG wire#powerrail
      Contact( "indexing_output_data".STEP11_MOTOR_90 )
   END_RUNG wire#w1
   // the same network as SCL:
   "STEPPER MOTOR 90°" := "indexing_output_data".STEP4_MOTOR_90 OR "indexing_output_data".STEP11_MOTOR_90;
END_REGION

REGION Network 5: indexing Gripper
   RUNG wire#powerrail
      Contact( "indexing_output_data"."close gripper" )
      Coil( "CLOSE GRIPPER 3A(1)" )
   END_RUNG
   RUNG wire#powerrail
      Contact( "indexing_output_data"."release gripper" )
      wire#w1
      Coil( "RELEASE GRIPPER 3A" )
   END_RUNG
   RUNG wire#powerrail
      Contact( "indexing_Modes_data".Reset )
   END_RUNG wire#w1
   // the same network as SCL:
   "CLOSE GRIPPER 3A(1)" := "indexing_output_data"."close gripper";
   "RELEASE GRIPPER 3A" := "indexing_output_data"."release gripper" OR "indexing_Modes_data".Reset;
END_REGION

REGION Network 6: indexing rotation Cylinder
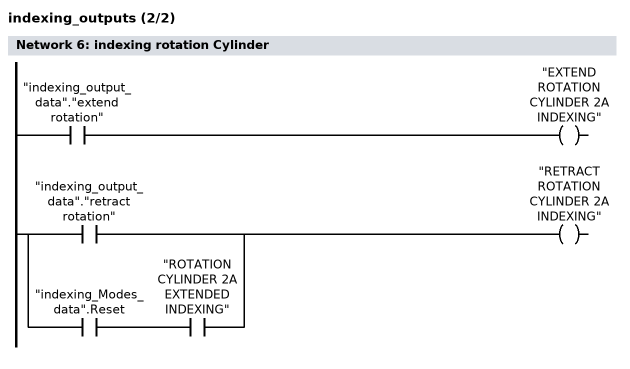
   RUNG wire#powerrail
      Contact( "indexing_output_data"."extend rotation" )
      Coil( "EXTEND ROTATION CYLINDER 2A INDEXING" )
   END_RUNG
   RUNG wire#powerrail
      Contact( "indexing_output_data"."retract rotation" )
      wire#w1
      Coil( "RETRACT ROTATION CYLINDER 2A INDEXING" )
   END_RUNG
   RUNG wire#powerrail
      Contact( "indexing_Modes_data".Reset )
      Contact( "ROTATION CYLINDER 2A EXTENDED INDEXING" )
   END_RUNG wire#w1
   // the same network as SCL:
   "EXTEND ROTATION CYLINDER 2A INDEXING" := "indexing_output_data"."extend rotation";
   "RETRACT ROTATION CYLINDER 2A INDEXING" := "indexing_output_data"."retract rotation" OR ("indexing_Modes_data".Reset AND "ROTATION CYLINDER 2A EXTENDED INDEXING");
END_REGION
END_FUNCTION

FUNCTION "indexing_operation" : Void   // FC7, LAD
{ S7_Optimized_Access := 'TRUE' }
VERSION : 0.1
   VAR_TEMP   // added for the SCL form of the ladder/FBD networks
      _w1 : Bool;
   END_VAR
BEGIN

REGION Network 1: STEP 1: Transfer from previous station
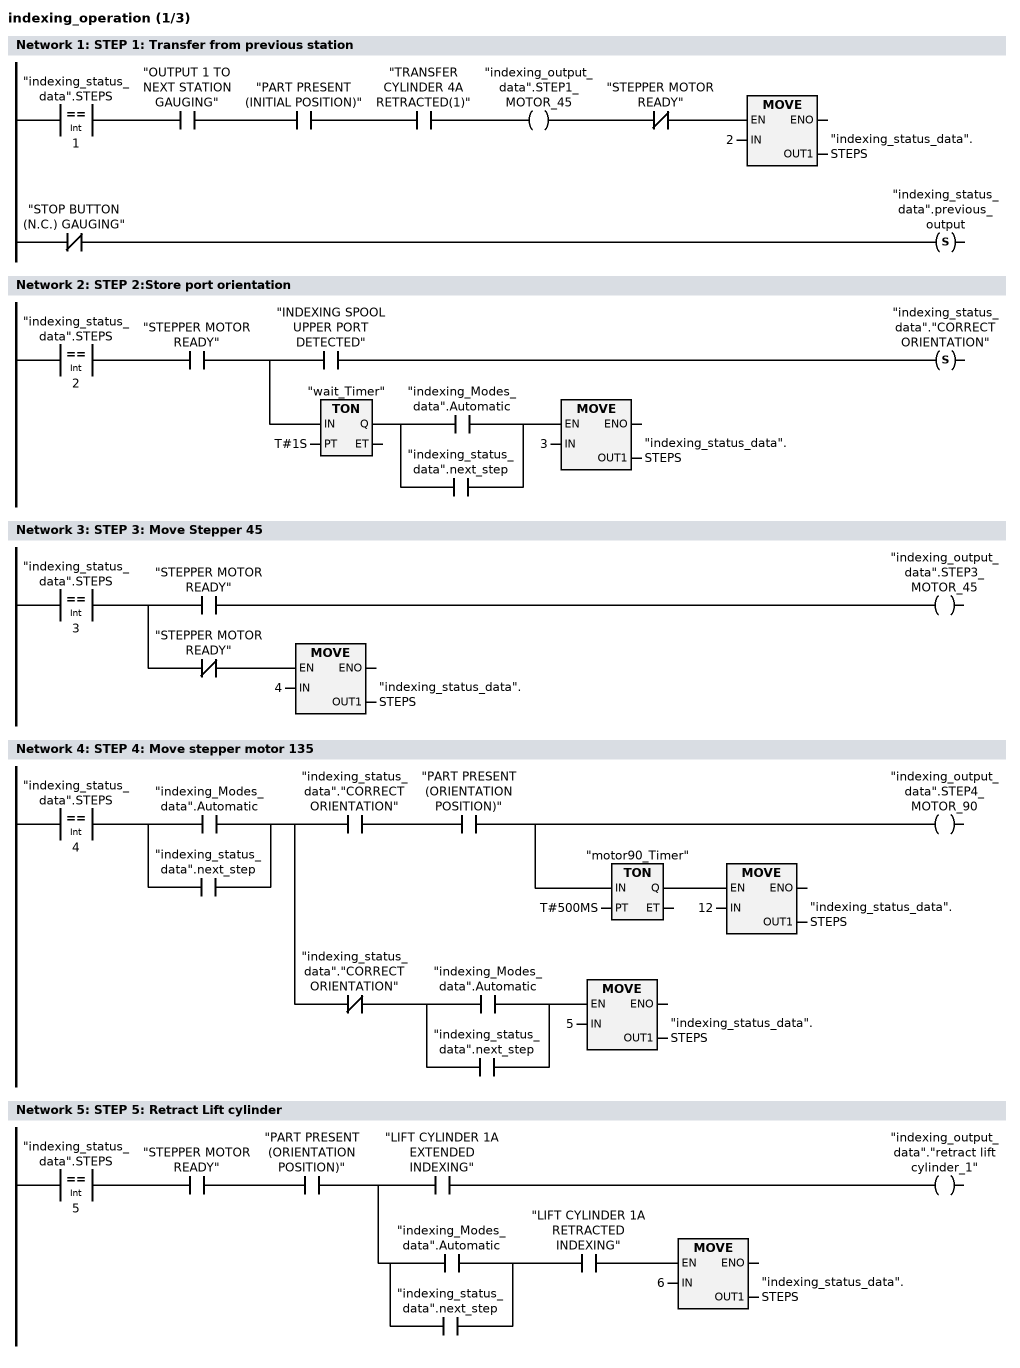
   RUNG wire#powerrail
      { S7_Templates := "SrcType := Int" } EQ_Contact(in1 := "indexing_status_data".STEPS, in2 := 1)
      Contact( "OUTPUT 1 TO NEXT STATION GAUGING" )
      Contact( "PART PRESENT (INITIAL POSITION)" )
      Contact( "TRANSFER CYLINDER 4A RETRACTED(1)" )
      Coil( "indexing_output_data".STEP1_MOTOR_45 )
      I_Contact( "STEPPER MOTOR READY" )
      Move(in := 2, out1 => "indexing_status_data".STEPS)
   END_RUNG
   RUNG wire#powerrail
      I_Contact( "STOP BUTTON (N.C.) GAUGING" )
      S_Coil( "indexing_status_data".previous_output )
   END_RUNG
   // the same network as SCL:
   "indexing_output_data".STEP1_MOTOR_45 := ("indexing_status_data".STEPS = 1) AND "OUTPUT 1 TO NEXT STATION GAUGING" AND "PART PRESENT (INITIAL POSITION)" AND "TRANSFER CYLINDER 4A RETRACTED(1)";
   IF "indexing_output_data".STEP1_MOTOR_45 AND NOT "STEPPER MOTOR READY" THEN
       "indexing_status_data".STEPS := 2;
   END_IF;
   IF NOT "STOP BUTTON (N.C.) GAUGING" THEN "indexing_status_data".previous_output := TRUE; END_IF;
END_REGION

REGION Network 2: STEP 2:Store port orientation
   #_w1 := ("indexing_status_data".STEPS = 2) AND "STEPPER MOTOR READY";
   IF #_w1 AND "INDEXING SPOOL UPPER PORT DETECTED" THEN
       "indexing_status_data"."CORRECT ORIENTATION" := TRUE;
   END_IF;
   "wait_Timer".TON(IN := #_w1, PT := T#1S);
   IF "wait_Timer".Q AND ("indexing_Modes_data".Automatic OR "indexing_status_data".next_step) THEN
       "indexing_status_data".STEPS := 3;
   END_IF;
END_REGION

REGION Network 3: STEP 3: Move Stepper 45
   RUNG wire#powerrail
      { S7_Templates := "SrcType := Int" } EQ_Contact(in1 := "indexing_status_data".STEPS, in2 := 3)
      wire#w1
      Contact( "STEPPER MOTOR READY" )
      Coil( "indexing_output_data".STEP3_MOTOR_45 )
   END_RUNG
   RUNG wire#w1
      I_Contact( "STEPPER MOTOR READY" )
      Move(in := 4, out1 => "indexing_status_data".STEPS)
   END_RUNG
   // the same network as SCL:
   #_w1 := "indexing_status_data".STEPS = 3;
   "indexing_output_data".STEP3_MOTOR_45 := #_w1 AND "STEPPER MOTOR READY";
   IF #_w1 AND NOT "STEPPER MOTOR READY" THEN "indexing_status_data".STEPS := 4; END_IF;
END_REGION

REGION Network 4: STEP 4: Move stepper motor 135
   #_w1 := ("indexing_status_data".STEPS = 4) AND ("indexing_Modes_data".Automatic OR "indexing_status_data".next_step);
   "indexing_output_data".STEP4_MOTOR_90 := #_w1 AND "indexing_status_data"."CORRECT ORIENTATION" AND "PART PRESENT (ORIENTATION POSITION)";
   "motor90_Timer".TON(IN := "indexing_output_data".STEP4_MOTOR_90, PT := T#500MS);
   IF "motor90_Timer".Q THEN "indexing_status_data".STEPS := 12; END_IF;
   IF #_w1 AND NOT "indexing_status_data"."CORRECT ORIENTATION" AND ("indexing_Modes_data".Automatic OR "indexing_status_data".next_step) THEN
       "indexing_status_data".STEPS := 5;
   END_IF;
END_REGION

REGION Network 5: STEP 5: Retract Lift cylinder
   RUNG wire#powerrail
      { S7_Templates := "SrcType := Int" } EQ_Contact(in1 := "indexing_status_data".STEPS, in2 := 5)
      Contact( "STEPPER MOTOR READY" )
      Contact( "PART PRESENT (ORIENTATION POSITION)" )
      wire#w1
      Contact( "LIFT CYLINDER 1A EXTENDED INDEXING" )
      Coil( "indexing_output_data"."retract lift cylinder_1" )
   END_RUNG
   RUNG wire#w1
      Contact( "indexing_Modes_data".Automatic )
      wire#w2
      Contact( "LIFT CYLINDER 1A RETRACTED INDEXING" )
      Move(in := 6, out1 => "indexing_status_data".STEPS)
   END_RUNG
   RUNG wire#w1
      Contact( "indexing_status_data".next_step )
   END_RUNG wire#w2
   // the same network as SCL:
   #_w1 := ("indexing_status_data".STEPS = 5) AND "STEPPER MOTOR READY" AND "PART PRESENT (ORIENTATION POSITION)";
   "indexing_output_data"."retract lift cylinder_1" := #_w1 AND "LIFT CYLINDER 1A EXTENDED INDEXING";
   IF #_w1 AND ("indexing_Modes_data".Automatic OR "indexing_status_data".next_step) AND "LIFT CYLINDER 1A RETRACTED INDEXING" THEN
       "indexing_status_data".STEPS := 6;
   END_IF;
END_REGION

REGION Network 6: STEP 6: CLOSE THE GRIPPER
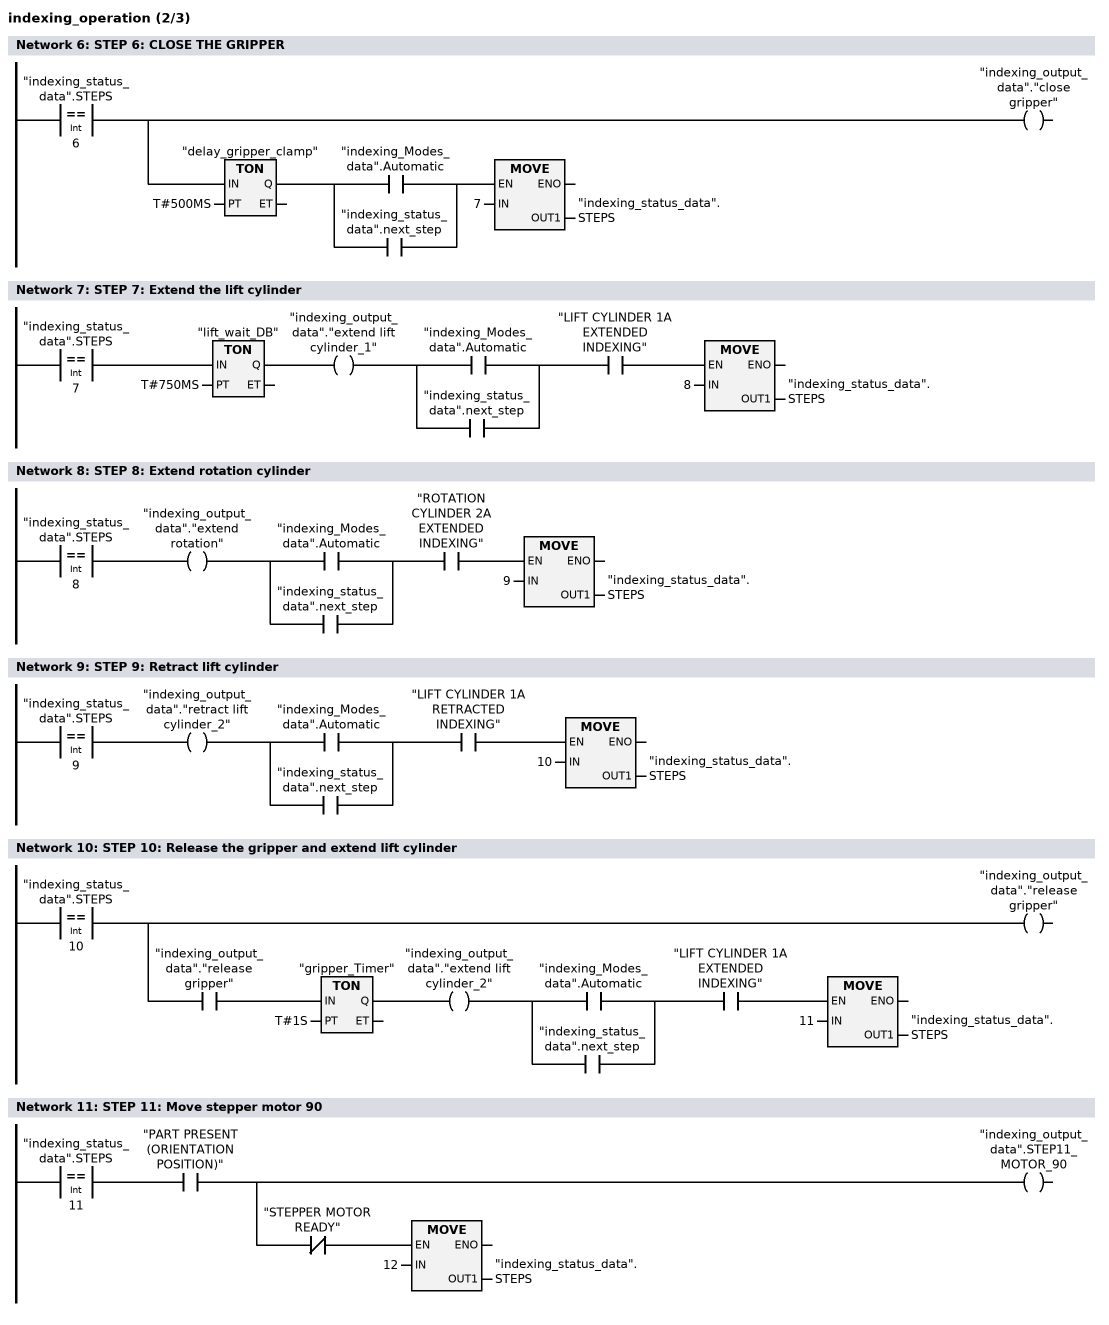
   "indexing_output_data"."close gripper" := "indexing_status_data".STEPS = 6;
   "delay_gripper_clamp".TON(IN := "indexing_output_data"."close gripper", PT := T#500MS);
   IF "delay_gripper_clamp".Q AND ("indexing_Modes_data".Automatic OR "indexing_status_data".next_step) THEN
       "indexing_status_data".STEPS := 7;
   END_IF;
END_REGION

REGION Network 7: STEP 7: Extend the lift cylinder
   "lift_wait_DB".TON(IN := "indexing_status_data".STEPS = 7, PT := T#750MS);
   "indexing_output_data"."extend lift cylinder_1" := "lift_wait_DB".Q;
   IF "lift_wait_DB".Q AND ("indexing_Modes_data".Automatic OR "indexing_status_data".next_step) AND "LIFT CYLINDER 1A EXTENDED INDEXING" THEN
       "indexing_status_data".STEPS := 8;
   END_IF;
END_REGION

REGION Network 8: STEP 8: Extend rotation cylinder
   RUNG wire#powerrail
      { S7_Templates := "SrcType := Int" } EQ_Contact(in1 := "indexing_status_data".STEPS, in2 := 8)
      Coil( "indexing_output_data"."extend rotation" )
      wire#w1
      Contact( "indexing_Modes_data".Automatic )
      wire#w2
      Contact( "ROTATION CYLINDER 2A EXTENDED INDEXING" )
      Move(in := 9, out1 => "indexing_status_data".STEPS)
   END_RUNG
   RUNG wire#w1
      Contact( "indexing_status_data".next_step )
   END_RUNG wire#w2
   // the same network as SCL:
   "indexing_output_data"."extend rotation" := "indexing_status_data".STEPS = 8;
   IF "indexing_output_data"."extend rotation" AND ("indexing_Modes_data".Automatic OR "indexing_status_data".next_step) AND "ROTATION CYLINDER 2A EXTENDED INDEXING" THEN
       "indexing_status_data".STEPS := 9;
   END_IF;
END_REGION

REGION Network 9: STEP 9: Retract lift cylinder
   RUNG wire#powerrail
      { S7_Templates := "SrcType := Int" } EQ_Contact(in1 := "indexing_status_data".STEPS, in2 := 9)
      Coil( "indexing_output_data"."retract lift cylinder_2" )
      wire#w1
      Contact( "indexing_Modes_data".Automatic )
      wire#w2
      Contact( "LIFT CYLINDER 1A RETRACTED INDEXING" )
      Move(in := 10, out1 => "indexing_status_data".STEPS)
   END_RUNG
   RUNG wire#w1
      Contact( "indexing_status_data".next_step )
   END_RUNG wire#w2
   // the same network as SCL:
   "indexing_output_data"."retract lift cylinder_2" := "indexing_status_data".STEPS = 9;
   IF "indexing_output_data"."retract lift cylinder_2" AND ("indexing_Modes_data".Automatic OR "indexing_status_data".next_step) AND "LIFT CYLINDER 1A RETRACTED INDEXING" THEN
       "indexing_status_data".STEPS := 10;
   END_IF;
END_REGION

REGION Network 10: STEP 10: Release the gripper and extend lift cylinder
   "indexing_output_data"."release gripper" := "indexing_status_data".STEPS = 10;
   "gripper_Timer".TON(IN := "indexing_output_data"."release gripper" AND "indexing_output_data"."release gripper",
                       PT := T#1S);
   "indexing_output_data"."extend lift cylinder_2" := "gripper_Timer".Q;
   IF "gripper_Timer".Q AND ("indexing_Modes_data".Automatic OR "indexing_status_data".next_step) AND "LIFT CYLINDER 1A EXTENDED INDEXING" THEN
       "indexing_status_data".STEPS := 11;
   END_IF;
END_REGION

REGION Network 11: STEP 11: Move stepper motor 90
   RUNG wire#powerrail
      { S7_Templates := "SrcType := Int" } EQ_Contact(in1 := "indexing_status_data".STEPS, in2 := 11)
      Contact( "PART PRESENT (ORIENTATION POSITION)" )
      wire#w1
      Coil( "indexing_output_data".STEP11_MOTOR_90 )
   END_RUNG
   RUNG wire#w1
      I_Contact( "STEPPER MOTOR READY" )
      Move(in := 12, out1 => "indexing_status_data".STEPS)
   END_RUNG
   // the same network as SCL:
   "indexing_output_data".STEP11_MOTOR_90 := ("indexing_status_data".STEPS = 11) AND "PART PRESENT (ORIENTATION POSITION)";
   IF "indexing_output_data".STEP11_MOTOR_90 AND NOT "STEPPER MOTOR READY" THEN
       "indexing_status_data".STEPS := 12;
   END_IF;
END_REGION

REGION Network 12: STEP 12: Extend Transfer Cylinder
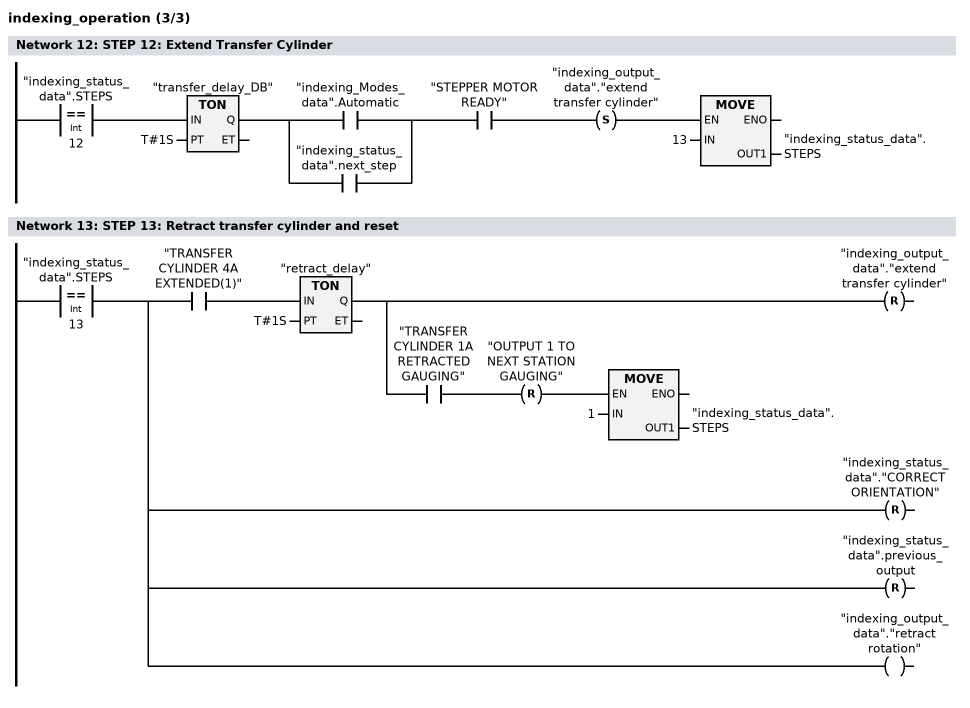
   "transfer_delay_DB".TON(IN := "indexing_status_data".STEPS = 12, PT := T#1S);
   IF "transfer_delay_DB".Q AND ("indexing_Modes_data".Automatic OR "indexing_status_data".next_step) AND "STEPPER MOTOR READY" THEN
       "indexing_output_data"."extend transfer cylinder" := TRUE;
       "indexing_status_data".STEPS := 13;
   END_IF;
END_REGION

REGION Network 13: STEP 13: Retract transfer cylinder and reset
   #_w1 := "indexing_status_data".STEPS = 13;
   "retract_delay".TON(IN := #_w1 AND "TRANSFER CYLINDER 4A EXTENDED(1)", PT := T#1S);
   IF "retract_delay".Q THEN "indexing_output_data"."extend transfer cylinder" := FALSE; END_IF;
   IF "retract_delay".Q AND "TRANSFER CYLINDER 1A RETRACTED GAUGING" THEN
       "OUTPUT 1 TO NEXT STATION GAUGING" := FALSE;
       "indexing_status_data".STEPS := 1;
   END_IF;
   IF #_w1 THEN
       "indexing_status_data"."CORRECT ORIENTATION" := FALSE;
       "indexing_status_data".previous_output := FALSE;
   END_IF;
   "indexing_output_data"."retract rotation" := #_w1;
END_REGION
END_FUNCTION

FUNCTION "indexing_utils" : Void   // FC8, LAD
{ S7_Optimized_Access := 'TRUE' }
VERSION : 0.1
BEGIN

REGION Network 1: SETUP: Start, reset
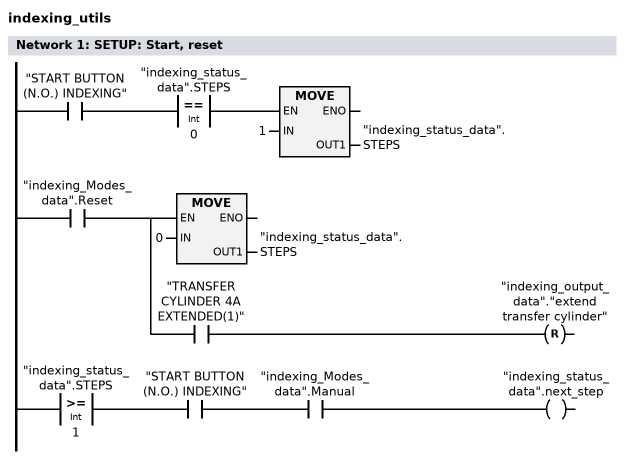
   RUNG wire#powerrail
      Contact( "START BUTTON  (N.O.) INDEXING" )
      { S7_Templates := "SrcType := Int" } EQ_Contact(in1 := "indexing_status_data".STEPS, in2 := 0)
      Move(in := 1, out1 => "indexing_status_data".STEPS)
   END_RUNG
   RUNG wire#powerrail
      Contact( "indexing_Modes_data".Reset )
      wire#w1
      Move(in := 0, out1 => "indexing_status_data".STEPS)
   END_RUNG
   RUNG wire#w1
      Contact( "TRANSFER CYLINDER 4A EXTENDED(1)" )
      R_Coil( "indexing_output_data"."extend transfer cylinder" )
   END_RUNG
   RUNG wire#powerrail
      { S7_Templates := "SrcType := Int" } GE_Contact(in1 := "indexing_status_data".STEPS, in2 := 1)
      Contact( "START BUTTON  (N.O.) INDEXING" )
      Contact( "indexing_Modes_data".Manual )
      Coil( "indexing_status_data".next_step )
   END_RUNG
   // the same network as SCL:
   IF "START BUTTON  (N.O.) INDEXING" AND ("indexing_status_data".STEPS = 0) THEN
       "indexing_status_data".STEPS := 1;
   END_IF;
   IF "indexing_Modes_data".Reset THEN "indexing_status_data".STEPS := 0; END_IF;
   IF "indexing_Modes_data".Reset AND "TRANSFER CYLINDER 4A EXTENDED(1)" THEN
       "indexing_output_data"."extend transfer cylinder" := FALSE;
   END_IF;
   "indexing_status_data".next_step := ("indexing_status_data".STEPS >= 1) AND "START BUTTON  (N.O.) INDEXING" AND "indexing_Modes_data".Manual;
END_REGION
END_FUNCTION

ORGANIZATION_BLOCK "Main"   // OB1, LAD, ProgramCycle
TITLE = "Main Program Sweep (Cycle)"
{ S7_Optimized_Access := 'TRUE' }
VERSION : 0.1
   VAR_INPUT
      Initial_Call : Bool;   // Initial call of this OB
      Remanence : Bool;   // =True, if remanent data are available
   END_VAR
BEGIN

REGION Network 1: Modes
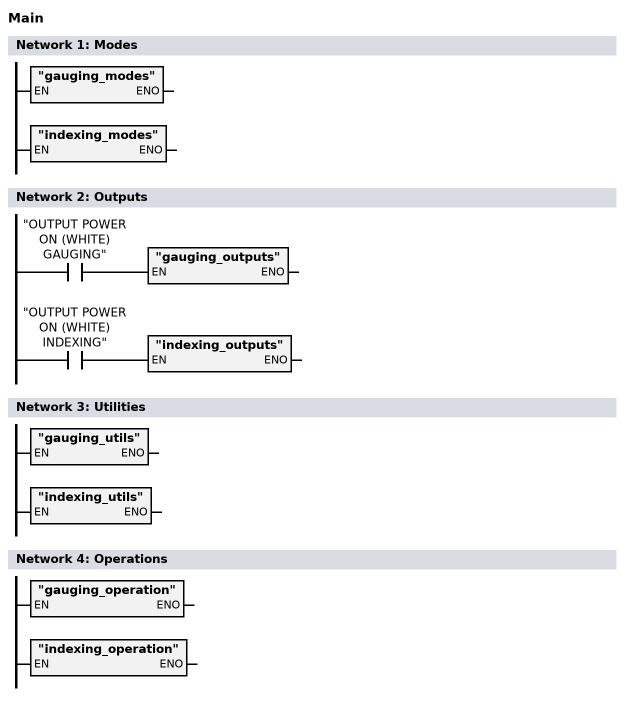
   RUNG wire#powerrail
      "gauging_modes"()
   END_RUNG
   RUNG wire#powerrail
      "indexing_modes"()
   END_RUNG
   // the same network as SCL:
   "gauging_modes"();
   "indexing_modes"();
END_REGION

REGION Network 2: Outputs
   RUNG wire#powerrail
      Contact( "OUTPUT POWER ON (WHITE) GAUGING" )
      "gauging_outputs"()
   END_RUNG
   RUNG wire#powerrail
      Contact( "OUTPUT POWER ON (WHITE) INDEXING" )
      "indexing_outputs"()
   END_RUNG
   // the same network as SCL:
   IF "OUTPUT POWER ON (WHITE) GAUGING" THEN "gauging_outputs"(); END_IF;
   IF "OUTPUT POWER ON (WHITE) INDEXING" THEN "indexing_outputs"(); END_IF;
END_REGION

REGION Network 3: Utilities
   RUNG wire#powerrail
      "gauging_utils"()
   END_RUNG
   RUNG wire#powerrail
      "indexing_utils"()
   END_RUNG
   // the same network as SCL:
   "gauging_utils"();
   "indexing_utils"();
END_REGION

REGION Network 4: Operations
   RUNG wire#powerrail
      "gauging_operation"()
   END_RUNG
   RUNG wire#powerrail
      "indexing_operation"()
   END_RUNG
   // the same network as SCL:
   "gauging_operation"();
   "indexing_operation"();
END_REGION
END_ORGANIZATION_BLOCK